RoboDK station: VSAT new robodk (nocontrol).rdk

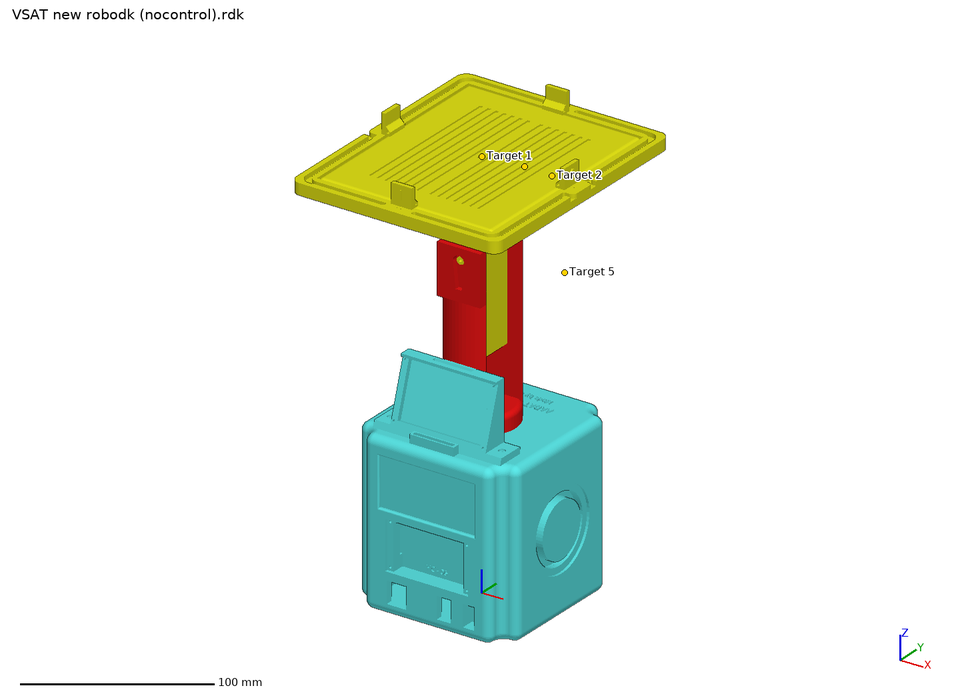
[picture v0: the station drawn from its stored meshes, robots at their saved joint values, targets as dots, program paths as lines]
Station AADAT new robodk (saved by RoboDK 5.5.3). Poses are relative to the parent item; angles as X-Y-Z fixed-axis rotations.
  - frame AADAT Base at (6.88, 1015.12, -100.97) mm
    - robot AADAT: 6 axes
        modified DH rows (alpha deg, a mm, theta deg, d mm): 0, 0, 0, 198; -90, 0, -90, 0; 0, 52, 0, 0; -90, 0, 0, 0; 90, 0, 0, 0; -90, 0, 180, 0
        joint limits [0, -90, 0, 0, 0, 0] to [180, 90, 0, 0, 0, 0]; home [0, 0, 0, 0, 0, 0]; saved at [0, 0, 0, 0, 0, 0]
    - target Target 1 (joint target) at (0, 0, 250) mm; joints [0, 0, 0, 0, 0, 0] of AADAT
    - target Target 2 (joint target) at (24.05, 28.66, 234.11) mm, rotated rx 0 ry 46.02 rz 50 deg; joints [50, 46.02, 0, 0, 0, 0] of AADAT
    - target Target 3 (joint target) at (-4.11, 44, 225.4) mm, rotated rx 0 ry 58.2 rz 95.33 deg; joints [95.33, 58.2, 0, 0, 0, 0] of AADAT
    - target Target 4 (joint target) at (0, 0, 250) mm; joints [0, 0, 0, 0, 0, 0] of AADAT
    - target Target 5 (joint target) at (52, 0, 198) mm, rotated rx 0 ry 90 rz 0 deg; joints [0, 90, 0, 0, 0, 0] of AADAT
  - Python program Single Pyserial Bluetooth (Excel)(NoControl)(OLED) (listed below)
  - Python program Dual Pyserial Bluetooth (Excel)(NoControl) (listed below)
  - Python program Single Pyserial Bluetooth (Excel)(Control)(OLED) (listed below)
  - Python program Dual Pyserial Bluetooth (Excel)(Control) (listed below)
  - Python program Coordinates (listed below)

--- Python program Single Pyserial Bluetooth (Excel)(NoControl)(OLED) ---
import time
import datetime
from openpyxl import *
import serial
port = 'COM11'
board = serial.Serial(port, 9600, timeout=10)

from robolink import *    # API to communicate with RoboDK
from robodk import *      # robodk robotics toolbox
# Any interaction with RoboDK must be done through RDK:
RDK = Robolink()

# get the robot by name:
robot = RDK.Item('', ITEM_TYPE_ROBOT)


def retrieveData():
    board.write(b'r')
    while board.inWaiting():
        pass
    data = board.readline().decode('ascii')
    return data

board.write(b'0')  # send 0 to arduino to reset angle to 90
time.sleep(1.1)

buffer_pos_vertical = 0
robot.setJoints([0,0,0,buffer_pos_vertical,0,0])      # set the robot movement's axes angle
row = 2

wb = Workbook()
ws = wb.active
ws.title = "Data"
ws.append(['Time', 'Date', 'ini_pos_v', 'Fin_LDR1', 'Fin_LDR3', 'Vo_Single(V)',
           'Vo_fixed(V)', 'Vin_Single(V)', 'Vin_fixed(V)', 'C_Single(mA)', 'C_fixed(mA)', 'P_Single(mW)',
           'P_fixed(mW)'])

while True:
    # joints = robot.Joints().list()
    data = retrieveData().strip('\r\n').split(',')
    print(data)
    #####################################################
    pos_vertical = int(data[0])
    robot_angle = pos_vertical - 90 #define new robot angle in robodk
    robot.setJoints([0,0,0,robot_angle,0,0])      # set the robot movement's axes angle
    light1 = int(data[1])
    light3 = int(data[2])
    real_Vo_Single = (float(data[3]))/1023 * 5
    real_Vo_Fixed = (float(data[4]))/1023 * 5
    C_Single = real_Vo_Single / 12250
    C_Fixed = real_Vo_Fixed / 12250
    Vin_Single = (C_Single * 22750) + real_Vo_Single
    Vin_Fixed = (C_Fixed * 22750) + real_Vo_Fixed
    P_Single = (pow(Vin_Single, 2)) / 35000
    P_Fixed = (pow(Vin_Fixed, 2)) / 35000
    ######################################################
    now = datetime.datetime.now()
    ws["A" + str(row)].value = now.strftime("%H:%M:%S")
    ws["B" + str(row)].value = now.strftime("%d/%m/%y")
    ws["C" + str(row)].value = pos_vertical
    ws["D" + str(row)].value = light1
    ws["E" + str(row)].value = light3
    ws["F" + str(row)].value = real_Vo_Single
    ws["G" + str(row)].value = real_Vo_Fixed
    ws["H" + str(row)].value = Vin_Single
    ws["I" + str(row)].value = Vin_Fixed
    ws["J" + str(row)].value = C_Single*1000
    ws["K" + str(row)].value = C_Fixed*1000
    ws["L" + str(row)].value = P_Single*1000
    ws["M" + str(row)].value = P_Fixed*1000
    wb.save(r"C:\Users\nkhai\Desktop\single_pyserial_Excel_NoControl(1).xlsx")
    ###########################################################
    row += 1
    time.sleep(1.1)
    # time.sleep(1200)

--- Python program Dual Pyserial Bluetooth (Excel)(NoControl) ---
import time
import datetime
from openpyxl import *
import serial
port = 'COM6'
board = serial.Serial(port, 9600, timeout=10)

from robolink import *    # API to communicate with RoboDK
from robodk import *      # robodk robotics toolbox
# from robodk.robomath import *
# Any interaction with RoboDK must be done through RDK:
RDK = Robolink()

# get the robot by name:
robot = RDK.Item('', ITEM_TYPE_ROBOT)


def retrieveData():
    board.write(b'r')
    while board.inWaiting():
        pass
    data = board.readline().decode('ascii')
    return data


board.write(b'0')  # send 0 to arduino to reset angle to 90
time.sleep(1.1)

buffer_pos_horizontal = -90 # home position in robodk
buffer_pos_vertical = 0 # home position in robodk
robot.setJoints([buffer_pos_horizontal,0,0,buffer_pos_vertical,0,0]) #reset the robot at robodk to home position
row = 2

wb = Workbook()
ws = wb.active
ws.title = "Data"
ws.append(['Time', 'Date', 'ini_pos_v', 'ini_pos_h', 'Fin_LDR1', 'Fin_LDR3', 'Fin_LDR2', 'Fin_LDR4', 'Vo_AADAT(V)',
           'Vo_fixed(V)', 'Vin_AADAT(V)', 'Vin_fixed(V)', 'C_AADAT(mA)', 'C_fixed(mA)', 'P_AADAT(mW)', 'P_fixed(mW)'])
while True:
    # Update()
    # pos_ref = robot.Pose()
    # print(pos_ref)
    # Joints(robot_item_list)
    # joints = robot.Joints().list()
    # print(joints)
    # SimulatorJoints()
    # JointPoses(joints=None)
    # JointsHome()
    # setJointsHome(joints)
    # getLink(type_linked=2)
    data = retrieveData().strip('\r\n').split(',')
    print(data)
#######################################################
    pos_vertical = int(data[0])
    pos_horizontal = int(data[1])
    robot_angle_vertical = pos_vertical - 90
    robot_angle_horizontal = pos_horizontal - 180
    robot.setJoints([robot_angle_horizontal,0,0,robot_angle_vertical,0,0])      # set the robot movement's axes angle
    avgtop = int(data[2])
    avgbot = int(data[3])
    avgleft = int(data[4])
    avgright = int(data[5])
    Vo_AADAT = (float(data[6]))*5/1023
    Vo_Fixed = (float(data[7]))*5/1023
    C_AADAT = Vo_AADAT/12250
    C_Fixed = Vo_Fixed/12250
    Vin_AADAT = (C_AADAT*22750)+Vo_AADAT
    Vin_Fixed = (C_Fixed*22750)+Vo_Fixed
    P_AADAT = pow(Vin_AADAT, 2)/35000
    P_Fixed = pow(Vin_Fixed, 2)/35000
    ######################################################
    now = datetime.datetime.now()
    ws["A" + str(row)].value = now.strftime("%H:%M:%S")
    ws["B" + str(row)].value = now.strftime("%d/%m/%y")
    ws["C" + str(row)].value = pos_vertical
    ws["D" + str(row)].value = pos_horizontal
    ws["E" + str(row)].value = avgtop
    ws["F" + str(row)].value = avgbot
    ws["G" + str(row)].value = avgleft
    ws["H" + str(row)].value = avgright
    ws["I" + str(row)].value = Vo_AADAT
    ws["J" + str(row)].value = Vo_Fixed
    ws["K" + str(row)].value = Vin_AADAT
    ws["L" + str(row)].value = Vin_Fixed
    ws["M" + str(row)].value = C_AADAT*1000
    ws["N" + str(row)].value = C_Fixed*1000
    ws["O" + str(row)].value = P_AADAT*1000
    ws["P" + str(row)].value = P_Fixed*1000
    wb.save(r'C:/Users/nkhai/Desktop/AADAT_pyserial_Excel_NoControl(Middle_Separate).xlsx')
    ###########################################################
    row += 1
    time.sleep(1.2)
    # time.sleep(300)

--- Python program Single Pyserial Bluetooth (Excel)(Control)(OLED) ---
import time
import datetime
import serial
from openpyxl import *
port = 'COM4'
board = serial.Serial(port, 9600, timeout=10)  # Change your port name COM... and your baudrate

from robolink import *    # API to communicate with RoboDK
from robodk import *      # robodk robotics toolbox
# Any interaction with RoboDK must be done through RDK:
RDK = Robolink()

# get the robot by name:
robot = RDK.Item('', ITEM_TYPE_ROBOT)


def retrieveData():
    board.write(b'r')
    while board.inWaiting():
        pass
    data = board.readline().decode('ascii')
    return data


def retrieveData_power():
    board.write(b'p')
    while board.inWaiting():
        pass
    data = board.readline().decode('ascii')
    return data


def vertical_up(pos):
    pos_v = pos
    range_d = 20
    range_n = -20
    while pos_v < 145:
        data = retrieveData().strip('\r\n').split(',')
        print(data)
        #########################################################
        light1 = int(data[0])
        light3 = int(data[1])
        pos_v = int(data[2])
        #########################################################
        if range_d > light1 - light3 > range_n:
            break
        elif (light1 - light3) < range_n:
            break
        else:
            pos_v += 1
            time.sleep(1.1)
            board.write(b'1')  # send 1 to arduino to increase the angle and let servo move
            robot_angle = pos_v - 90 #define new robot angle in robodk
            robot.setJoints([0,0,0,robot_angle,0,0])      # set the robot movement's axes angle
            time.sleep(1.1)
    time.sleep(1.1)
    return pos_v


def vertical_down(pos):
    pos_v = pos
    range_d = 20
    range_n = -20
    while pos_v > 35:
        data = retrieveData().strip('\r\n').split(',')
        print(data)
        #########################################################
        light1 = int(data[0])
        light3 = int(data[1])
        pos_v = int(data[2])
        #########################################################
        if range_d > light1 - light3 > range_n:
            break
        elif (light1 - light3) > range_d:
            break
        else:
            pos_v -= 1
            time.sleep(1.1)
            board.write(b'2')  # send 2 to arduino to decrease the angle and let servo move
            robot_angle = pos_v - 90 #define new robot angle in robodk
            robot.setJoints([0,0,0,robot_angle,0,0])      # set the robot movement's axes angle
            time.sleep(1.1)
    time.sleep(1.1)
    return pos_v


board.write(b'0')  # send 0 to arduino to reset angle to 90
time.sleep(1.1)

range_difference = 20
range_negative = -20
pos_vertical = 90
buffer_pos_vertical = 0
robot.setJoints([0,0,0,buffer_pos_vertical,0,0])      #reset robot at robodk to home position
row = 2

wb = Workbook()
ws = wb.active
ws.title = "Data"
ws.append(['Time', 'Date', 'ini_pos_v', 'Fin_LDR1', 'Fin_LDR3', 'VIn_Single(V)', 'VIn_fixed(V)',
           'Vin_Single(V)', 'Vin_fixed(V)', 'C_Single(mA)', 'C_fixed(mA)', 'P_Single(mW)', 'P_fixed(mW)'])

while True:
    # joints = robot.Joints().list()
    data = retrieveData().strip('\r\n').split(',')
    print(data)
    time.sleep(1.1)
    light1 = int(data[0])
    light3 = int(data[1])
    pos_vertical = int(data[2])
    #########################################################
    if (light1 - light3) > range_difference:
        pos_vertical = vertical_up(pos_vertical)
    if (light1 - light3) < range_negative:
        pos_vertical = vertical_down(pos_vertical)
#########################################################
    power_data = retrieveData_power().strip('\r\n').split(',')  # read data from arduino
    Vo_Single = float(power_data[0])*5/1023
    Vo_Fixed = float(power_data[1])*5/1023
    C_Single = Vo_Single / 12250
    C_Fixed = Vo_Fixed / 12250
    Vin_Single = (C_Single * 22750) + Vo_Single
    Vin_Fixed = (C_Fixed * 22750) + Vo_Fixed
    P_Single = pow(Vin_Single, 2) / 35000
    P_Fixed = pow(Vin_Fixed, 2) / 35000
#########################################################
    now = datetime.datetime.now()
    ws["A" + str(row)].value = now.strftime("%H:%M:%S")
    ws["B" + str(row)].value = now.strftime("%d/%m/%y")
    ws["C" + str(row)].value = pos_vertical
    ws["D" + str(row)].value = light1
    ws["E" + str(row)].value = light3
    ws["F" + str(row)].value = Vo_Single
    ws["G" + str(row)].value = Vo_Fixed
    ws["H" + str(row)].value = Vin_Single
    ws["I" + str(row)].value = Vin_Fixed
    ws["J" + str(row)].value = C_Single*1000
    ws["K" + str(row)].value = C_Fixed*1000
    ws["L" + str(row)].value = P_Single*1000
    ws["M" + str(row)].value = P_Fixed*1000
    wb.save(r"C:\Users\nkhai\Desktop\single_pyserial_Excel_Control.xlsx")
    ###########################################################
    row += 1
    time.sleep(1.1)

--- Python program Dual Pyserial Bluetooth (Excel)(Control) ---
import time
import datetime
import serial
from openpyxl import *
port = 'COM10'
board = serial.Serial(port, 9600, timeout=10)  # Change your port name COM... and your baudrate

from robolink import *    # API to communicate with RoboDK
from robodk import *      # robodk robotics toolbox
# Any interaction with RoboDK must be done through RDK:
RDK = Robolink()

# get the robot by name:
robot = RDK.Item('', ITEM_TYPE_ROBOT)


def retrieveData13():
    board.write(b'r')
    while board.inWaiting():
        pass
    data = board.readline().decode('ascii')
    return data


def retrieveData24():
    board.write(b'q')
    while board.inWaiting():
        pass
    data = board.readline().decode('ascii')
    return data


def retrieveData_power():
    board.write(b'p')
    while board.inWaiting():
        pass
    data = board.readline().decode('ascii')
    return data


def horizontal_right(pos2):
    pos_h = pos2
    range_d = 20
    range_n = -20
    while pos_h < 180:
        data = retrieveData24().strip('\r\n').split(',')
        print(data)
        #########################################################
        light2 = int(data[0])
        light4 = int(data[1])
        pos_v = int(data[2])
        pos_h = int(data[3])
        #########################################################
        if range_d > light4 - light2 > range_n:
            break
        elif pos_v > 90:
            if light4 - light2 < range_n:
                break
        else:  # pos<=90
            if light4 - light2 > range_d:
                break
        pos_h += 1
        time.sleep(1.1)
        board.write(b'3')
        robot_angle_vertical = pos_v - 90
        robot_angle_horizontal = pos_h - 180
        robot.setJoints([robot_angle_horizontal,0,0,robot_angle_vertical,0,0])      # set the robot movement's axes angle
        time.sleep(1.1)
    time.sleep(1.1)
    return pos_h


def horizontal_left(pos2):
    pos_h = pos2
    range_d = 20
    range_n = -20
    while pos_h > 0:
        data = retrieveData24().strip('\r\n').split(',')
        print(data)
        #########################################################
        light2 = int(data[0])
        light4 = int(data[1])
        pos_v = int(data[2])
        pos_h = int(data[3])
        #########################################################
        if range_d > light4 - light2 > range_n:
            break
        elif pos_v > 90:
            if light4 - light2 > range_d:
                break
        else:  # pos<=90
            if light4 - light2 < range_n:
                break
        pos_h -= 1
        time.sleep(1.1)
        board.write(b'4')
        robot_angle_vertical = pos_v - 90
        robot_angle_horizontal = pos_h - 180
        robot.setJoints([robot_angle_horizontal,0,0,robot_angle_vertical,0,0])      # set the robot movement's axes angle
        time.sleep(1.1)
    time.sleep(1.1)
    return pos_h


def vertical_up(pos,buffer_pos_horizontal):
    pos_v = pos
    range_d = 20
    range_n = -20
    while pos_v < 145:
        data = retrieveData13().strip('\r\n').split(',')
        print(data)
        #########################################################
        light1 = int(data[0])
        light3 = int(data[1])
        pos_v = int(data[2])
        #########################################################
        if range_d > light1 - light3 > range_n:
            break
        elif (light1 - light3) < range_n:
            break
        else:
            pos_v += 1
            time.sleep(1.1)
            board.write(b'1')  # send 1 to arduino to increase the angle and let servo move
            robot_angle_vertical = pos_v - 90 #define new robot angle in robodk
            robot.setJoints([buffer_pos_horizontal,0,0,robot_angle_vertical,0,0])      # set the robot movement's axes angle
            time.sleep(1.1)
    time.sleep(1.1)
    return pos_v


def vertical_down(pos,buffer_pos_horizontal):
    pos_v = pos
    range_d = 20
    range_n = -20
    while pos_v > 35:
        data = retrieveData13().strip('\r\n').split(',')
        print(data)
        #########################################################
        light1 = int(data[0])
        light3 = int(data[1])
        pos_v = int(data[2])
        #########################################################
        if range_d > light1 - light3 > range_n:
            break
        elif (light1 - light3) > range_d:
            break
        else:
            pos_v -= 1
            time.sleep(1.1)
            board.write(b'2')  # send 2 to arduino to decrease the angle and let servo move
            robot_angle_vertical = pos_v - 90 #define new robot angle in robodk
            robot.setJoints([buffer_pos_horizontal,0,0,robot_angle_vertical,0,0])      # set the robot movement's axes angle
            time.sleep(1.1)
    time.sleep(1.1)
    return pos_v


board.write(b'0')  # send 0 to arduino to reset angle to 90
time.sleep(1.1)

range_difference = 20
range_negative = -20
buffer_pos_horizontal = -90 #home position in robodk
buffer_pos_vertical = 0 #home position in robodk
robot.setJoints([buffer_pos_horizontal,0,0,buffer_pos_vertical,0,0]) #reset the robot at robodk to home position

row = 2

wb = Workbook()
ws = wb.active
ws.title = "Data"
ws.append(['Time', 'Date', 'ini_pos_v', 'ini_pos_h', 'Fin_LDR1', 'Fin_LDR3', 'Fin_LDR2', 'Fin_LDR4', 'Vo_AADAT(V)',
           'Vo_fixed(V)', 'Vin_AADAT(V)', 'Vin_fixed(V)', 'C_AADAT(mA)', 'C_fixed(mA)', 'P_AADAT(mW)', 'P_fixed(mW)'])

while True:
    # joints = robot.Joints().list()
    data = retrieveData13().strip('\r\n').split(',')
    print(data)
    time.sleep(1.1)
    light1 = int(data[0])
    light3 = int(data[1])
    pos_vertical = int(data[2])
#########################################################
    if (light1 - light3) > range_difference:
        pos_vertical = vertical_up(pos_vertical,buffer_pos_horizontal)
    if (light1 - light3) < range_negative:
        pos_vertical = vertical_down(pos_vertical,buffer_pos_horizontal)
#########################################################
    data = retrieveData24().strip('\r\n').split(',')
    print(data)
    time.sleep(1.1)
    light2 = int(data[0])
    light4 = int(data[1])
    pos_vertical = int(data[2])
    pos_horizontal = int(data[3])
#########################################################
    if (light4 - light2) > range_difference:
        if pos_vertical > 90:
            pos_horizontal = horizontal_right(pos_horizontal)
        else:
            pos_horizontal = horizontal_left(pos_horizontal)
#########################################################
    if (light4 - light2) < range_negative:
        if pos_vertical > 90:
            pos_horizontal = horizontal_left(pos_horizontal)
        else:
            pos_horizontal = horizontal_right(pos_horizontal)
    buffer_pos_horizontal = pos_horizontal
#########################################################
    power_data = retrieveData_power().strip('\r\n').split(',')  # read data from arduino
    Vo_AADAT = float(power_data[0])*5/1023
    Vo_Fixed = float(power_data[1])*5/1023
    C_AADAT = Vo_AADAT / 12250
    C_Fixed = Vo_Fixed / 12250
    Vin_AADAT = (C_AADAT * 22750) + Vo_AADAT
    Vin_Fixed = (C_Fixed * 22750) + Vo_Fixed
    P_AADAT = pow(Vin_AADAT, 2) / 35000
    P_Fixed = pow(Vin_Fixed, 2) / 35000
#########################################################
    now = datetime.datetime.now()
    ws["A" + str(row)].value = now.strftime("%H:%M:%S")
    ws["B" + str(row)].value = now.strftime("%d/%m/%y")
    ws["C" + str(row)].value = pos_vertical
    ws["D" + str(row)].value = pos_horizontal
    ws["E" + str(row)].value = light1
    ws["F" + str(row)].value = light3
    ws["G" + str(row)].value = light2
    ws["H" + str(row)].value = light4
    ws["I" + str(row)].value = Vo_AADAT
    ws["J" + str(row)].value = Vo_Fixed
    ws["K" + str(row)].value = Vin_AADAT
    ws["L" + str(row)].value = Vin_Fixed
    ws["M" + str(row)].value = C_AADAT*1000
    ws["N" + str(row)].value = C_Fixed*1000
    ws["O" + str(row)].value = P_AADAT*1000
    ws["P" + str(row)].value = P_Fixed*1000
    wb.save(r"C:\Users\nkhai\Desktop\AADAT_pyserial_Excel_Control.xlsx")
    ###########################################################
    row += 1
    time.sleep(1.1)

--- Python program Coordinates ---
# Type help("robodk.robolink") or help("robodk.robomath") for more information
# Press F5 to run the script
# Documentation: https://robodk.com/doc/en/RoboDK-API.html
# Reference:     https://robodk.com/doc/en/PythonAPI/robodk.html
# Note: It is not required to keep a copy of this file, your Python script is saved with your RDK project

import math
pi = 3.14159265359
# You can also use the new version of the API:
from robodk import robolink    # RoboDK API
from robodk import robomath    # Robot toolbox
RDK = robolink.Robolink()

# Forward and backwards compatible use of the RoboDK API:
# Remove these 2 lines to follow python programming guidelines
from robodk import *      # RoboDK API
from robolink import *    # Robot toolbox
# Link to RoboDK
# RDK = Robolink()

# Any interaction with RoboDK must be done through RDK:
RDK = Robolink()

# get the robot by name:
robot = RDK.Item('', ITEM_TYPE_ROBOT)
while True:
    xyz_coordinate = input("Enter xyz coordinates with no space:\n").split(',')
    print(xyz_coordinate)
    x = float(xyz_coordinate[0])
    y = float(xyz_coordinate[1])
    z = float(xyz_coordinate[2])
    print(x)
    print(y)
    print(z)
    pos1 = round(math.atan(y/x)*180/pi);
    if x<0:
        pos1 = round(math.atan(y/abs(x))*180/pi);
        pos1 = 180 - pos1;
    h = math.sqrt(x*x+y*y);
    pos2 = 90 - (round(math.atan((z-198)/h)*180/pi));
    robot.setJoints([pos1,pos2,0,0,0,0])      # set the robot movement's axes angle
